(* CODESYS project 2019-30-07-Sparkplug_Commands.ecp

Project tree, tasks and I/O mapping:
  PFC_Sparkplug : 750-8212 PFC200 2ETH RS, WAGO, order no. 0750-8212, version 5.13.2.32
    application Application
      libraries: ; WagoAppCloud, 1.3.0.8 (WAGO)
      task PLC_Task (cyclic, interval t#100ms, priority 15) calls PLC_PRG
      program PLC_PRG [ST]
      program VariableLogger [ST]
      program CommandHandler [ST]
      function block FbChangeOfValue_Real [ST]
      function block FbChangeOfValue_Byte [ST]
      function block FbChangeOfValue_Bool [ST]
    Kbus : Kbus, WAGO, version 1.4.0.2
        unmapped channels: K-BUS diagnostics
    MODBUS
      MODBUS : MODBUS, WAGO, order no. n/a, version 1.1.1.15
    Serial
      COM1 : COM1, WAGO, version 0.0.0.19
    Common.PCI
*)

// PFC_Sparkplug/Application/PLC_PRG
(* Purpose of the example program: Communicate with a Sparkplug primary application *)
PROGRAM PLC_PRG

CommandHandler();
VariableLogger();

END_PROGRAM

// PFC_Sparkplug/Application/CommandHandler
(* Purpose of the example program: Receive and handle commands aka "metric-change-requests" from the Sparkplug primary application
Ignition has functionality for "write tag", so within the commands our example program will define exacly one parameter,
which is actually the writable metric from ignitions point of view. 
The data protocol Sparkplug doesn't support response messages. (FbCommandResponse) *)
PROGRAM CommandHandler
VAR
	(* Use the function block FbCommandConfigurator to send the command configuration to the cloud *)
	oFbCmdConfigurator : 	WagoAppCloud.FbCommandConfigurator;
	(* Define two commands in the list *)
	aCommandDescriptions : 	ARRAY [0..1] OF WagoAppCloud.typCommandDescription;

	(*	Listen to command calls from the cloud using the FbCommandListener.
	It will set the xCommandReceived flag to true if a command is called. *)
	oFbCmdHandler : WagoAppCloud.FbCommandListener;
	xCommandReceived: BOOL;
	IncomingCommand : WagoAppCloud.typCommandRequest;
	dwReceivedCmdId : DWORD;

	(* Parameter to get the received value from the cloud *)
	rParameter1 : REAL;
	sParameter2 : STRING;
END_VAR

(* Init command1 and its Request Parameter *)		
aCommandDescriptions[0].bCommandId := 1;
aCommandDescriptions[0].bNumberOfRequestParameters := 1;
aCommandDescriptions[0].bNumberOfResponseParameters := 0;	(* The data protocol Sparkplug doesn't support response messages. This is an information for Wago Protocol. *)
aCommandDescriptions[0].sName := 'MyFirstCommand';
aCommandDescriptions[0].aRequestParameters[0].sParameterName := 'Parameter 1 from Cloud to PFC';
aCommandDescriptions[0].aRequestParameters[0].eParameterType := WagoAppCloud.eCommandParameterType.CPT_REAL;

(* Init command2 and its Request Parameter *)		
aCommandDescriptions[1].bCommandId := 2;
aCommandDescriptions[1].bNumberOfRequestParameters := 1;
aCommandDescriptions[1].bNumberOfResponseParameters := 0;
aCommandDescriptions[1].sName := 'MySecondCommand';
aCommandDescriptions[1].aRequestParameters[0].sParameterName := 'Parameter 2 from Cloud to PFC';
aCommandDescriptions[1].aRequestParameters[0].eParameterType := WagoAppCloud.eCommandParameterType.CPT_STRING;

(* Configurate the commands and send the commands configuration to the cloud *)
oFbCmdConfigurator(	pSupportedCommands := ADR(aCommandDescriptions),
					bNumberOfSupportedCommands := 2);

(* Receive data to get the command from the cloud *)
oFbCmdHandler(pCommand:= ADR(IncomingCommand), 
				xCommandReceived=> xCommandReceived);

(* Handle command *)
IF xCommandReceived THEN
	dwReceivedCmdId := IncomingCommand.dwCommandId;

	CASE dwReceivedCmdId OF
		1:
			(* received command with the command ID 1 *)
			rParameter1 := STRING_TO_REAL(IncomingCommand.aRequestParameters[0].sParameterValue);
			
		2:
			(* received command with the command ID 2 *)
			sParameter2 := IncomingCommand.aRequestParameters[0].sParameterValue;
	END_CASE
END_IF

END_PROGRAM

// PFC_Sparkplug/Application/VariableLogger
PROGRAM VariableLogger

VAR
	(* Some value to transfer *)
	iVariable1 		: INT 	:= -32768;
	dwVariable2		: DWORD := 7;
	lrVariable3		: LREAL	:= 21.53;

	bVariable4		: BYTE 	:= 255;
	xVariable5		: BOOL := FALSE;
	rVariable6		: REAL 	:= 1.234;	
	
	wVariable7		: WORD	:= 49;
	iVariable8		: INT 	:= -32768;
	
	(* Define 3 collections *)
	aCollections	: ARRAY[0..2] OF WagoAppCloud.typCollection;

	(* Define 3 variable descriptions for the collections *)
	aVariableDescriptions1	: ARRAY[0..2] OF WagoAppCloud.typVariableDescription;
	aVariableDescriptions2	: ARRAY[0..2] OF WagoAppCloud.typVariableDescription;
	aVariableDescriptions3	: ARRAY[0..1] OF WagoAppCloud.typVariableDescription;
	
	tSampleInterval1		: TIME := T#10S;
	tMinPublishInterval		: TIME := T#0S; (* choose the smallest possible publish interval *)
	
	oFbCollectionLogger		: WagoAppCloud.FbCollectionLogger;
END_VAR

VAR
	oFbChangeOfValue		: FbChangeOfValue_Bool;
	oFbChangeOfValue_Real	: FbChangeOfValue_Real;
	oFbChangeOfValue_Byte	: FbChangeOfValue_Byte;
	
	(* Timer *)
	xEnableTimer: BOOL := TRUE;
	tCyclicTimerSendTagCollection: TON;
END_VAR

(* Simulate changing values to transfer to the cloud *)
	iVariable1 := iVariable1 + 3;
	dwVariable2 := dwVariable2 + 100;
	lrVariable3 := lrVariable3 - 1234.12;
	bVariable4 := bVariable4 + 2;
	IF bVariable4 > 150 THEN
		xVariable5 := TRUE;
	ELSE
		xVariable5 := FALSE;
	END_IF
	rVariable6 := rVariable6 + 100;
	wVariable7 := wVariable7 + 1;
	iVariable8 := iVariable8 + 1;

(* Configuration of the collections and variables *)
	
(* Init and configure collection 1 *)
	aVariableDescriptions1[0].pAddress := ADR(iVariable1);
	aVariableDescriptions1[0].eValueType := WagoAppCloud.VVT_INT;
	aVariableDescriptions1[0].sTag := 'var1_int';
	aVariableDescriptions1[0].sUnit := 'u1';
	
	aVariableDescriptions1[1].pAddress := ADR(dwVariable2);
	aVariableDescriptions1[1].eValueType := WagoAppCloud.VVT_DWORD;
	aVariableDescriptions1[1].sTag := 'var2_dword';
	aVariableDescriptions1[1].sUnit := 'u2';
	
	aVariableDescriptions1[2].pAddress := ADR(lrVariable3);
	aVariableDescriptions1[2].eValueType := WagoAppCloud.VVT_LREAL;
	aVariableDescriptions1[2].sTag := 'var3_lreal';
	aVariableDescriptions1[2].sUnit := 'u3';
	
	aCollections[0].dwCollectionId := 1;
	aCollections[0].sName := 'MyFirstCollection';
	aCollections[0].pVariableDescriptions := ADR(aVariableDescriptions1);
	aCollections[0].dwVariablesCount := 3;
	(* Configuration of the mode to sampling the data. 
	In this case the samples of collection 1 will be set automatically. The space between two timestamps are defined in the sample interval. *)
	aCollections[0].eSamplingDataMode := eSamplingMode.LIBRARY_DEFAULT_AUTOMATIC;		(* LIBRARY_DEFAULT_AUTOMATIC is the default mode *)
	aCollections[0].pSampleInterval := ADR(tSampleInterval1);
	aCollections[0].pPublishInterval := ADR(tMinPublishInterval);

(* Init and configure collection 2 *)
	aVariableDescriptions2[0].pAddress := ADR(bVariable4);
	aVariableDescriptions2[0].eValueType := WagoAppCloud.VVT_BYTE;
	aVariableDescriptions2[0].sTag := 'var4_byte';
	aVariableDescriptions2[0].sUnit := 'u3';
	
	aVariableDescriptions2[1].pAddress := ADR(xVariable5);
	aVariableDescriptions2[1].eValueType := WagoAppCloud.VVT_BOOL;
	aVariableDescriptions2[1].sTag := 'var5_bool';
	aVariableDescriptions2[1].sUnit := 'u4';
	
	aVariableDescriptions2[2].pAddress := ADR(rVariable6);
	aVariableDescriptions2[2].eValueType := WagoAppCloud.VVT_REAL;
	aVariableDescriptions2[2].sTag := 'var6_real';
	aVariableDescriptions2[2].sUnit := 'u5';
	
	aCollections[1].dwCollectionId := 2;
	aCollections[1].sName := 'MySecondCollection';
	aCollections[1].pVariableDescriptions := ADR(aVariableDescriptions2);
	aCollections[1].dwVariablesCount := 3;
	(* Configuration of the mode to sampling the data. 
	In this case the samples of collection 2 will be set manual by the PLC application. 
	The Trigger of a sample is set manual with the CollectionTrigger or the VariableTrigger.
	
	Note for data protocol Sparkplug: The sampling mode UNEQUALLY_SPACED_CUSTOMIZED_SAMPLES will be used for all manual generatted samples. 
	Sampling modes UNEQUALLY_SPACED_COLLECTION_SAMPLES, EQUALLY_SPACED_COLLECTION_SAMPLES, EQUALLY_SPACED_CUSTOMIZED_SAMPLES are not needed for Sparkplug. 
	This differentation between the different manual generatted sample modes is only an interesting information for the Wago Protocol. *)
	aCollections[1].eSamplingDataMode := eSamplingMode.UNEQUALLY_SPACED_CUSTOMIZED_SAMPLES; 
	aCollections[1].pPublishInterval := ADR(tMinPublishInterval);
	
(* Init and cnfigure collection 3 *)
	aVariableDescriptions3[0].pAddress := ADR(wVariable7);
	aVariableDescriptions3[0].eValueType := WagoAppCloud.VVT_WORD;
	aVariableDescriptions3[0].sTag := 'var7_word';
	aVariableDescriptions3[0].sUnit := 'u3';
	
	aVariableDescriptions3[1].pAddress := ADR(iVariable8);
	aVariableDescriptions3[1].eValueType := WagoAppCloud.VVT_INT;
	aVariableDescriptions3[1].sTag := 'var8_int';
	aVariableDescriptions3[1].sUnit := 'u4';
	
	aCollections[2].dwCollectionId := 3;
	aCollections[2].sName := 'MyThirdCollection';
	aCollections[2].pVariableDescriptions := ADR(aVariableDescriptions3);
	aCollections[2].dwVariablesCount := 2;
	(* Configuration of the mode to sampling the data. 
	In this case the samples of collection 3 will be set manual by the PLC application. 
	The Trigger of a sample is set manual with the CollectionTrigger or the VariableTrigger. 
	
	Note for data protocol Sparkplug: The sampling mode UNEQUALLY_SPACED_CUSTOMIZED_SAMPLES will be used for all manual generatted samples. 
	Sampling modes UNEQUALLY_SPACED_COLLECTION_SAMPLES, EQUALLY_SPACED_COLLECTION_SAMPLES, EQUALLY_SPACED_CUSTOMIZED_SAMPLES are not needed for Sparkplug. 
	This differentation between the different manual generatted sample modes is only an interesting information for the Wago Protocol. *)
	aCollections[2].eSamplingDataMode := eSamplingMode.UNEQUALLY_SPACED_CUSTOMIZED_SAMPLES;
	aCollections[2].pPublishInterval := ADR(tMinPublishInterval);

(* Example to set the event if variable value exceeded the threshold values - Variable Trigger*)
oFbChangeOfValue_Byte(	bInput:= bVariable4,
						bActivate:= 100,
						bDeactivate:= 70,
						xTrigger:= aVariableDescriptions2[0].xVariableTrigger);

oFbChangeOfValue(	xVariable:= xVariable5, 
					xTrigger:= aVariableDescriptions2[1].xVariableTrigger);

oFbChangeOfValue_Real(	rInput:= rVariable6, 
						rActivate:= 1500,
						rDeactivate:= 700,
						xTrigger:= aVariableDescriptions2[2].xVariableTrigger);

(* Example to set the event with a timer intervall - CollectionTrigger or VariableTrigger *)
(* Set an event with an Timer to send the variables in an intervall to the cloud *)
tCyclicTimerSendTagCollection(IN:= xEnableTimer, PT:= T#30S);

IF tCyclicTimerSendTagCollection.Q THEN
	aCollections[1].xCollectionTrigger := TRUE;
	aCollections[2].xCollectionTrigger := TRUE;

	xEnableTimer := FALSE;
ELSE
	xEnableTimer := TRUE;
END_IF
						
oFbCollectionLogger(pCollections := ADR(aCollections),
					dwCollectionsCount := 3);

END_PROGRAM

// PFC_Sparkplug/Application/FbChangeOfValue_Bool
FUNCTION_BLOCK FbChangeOfValue_Bool
VAR_INPUT
	xVariable : BOOL; 	(* Input value *)
END_VAR
VAR_IN_OUT
	xTrigger : BOOL; 	(* Variable Trigger - trigger is set only once when the value was changed and reset with the function block WagoAppCloud.FbCollectionLogger *)
END_VAR
VAR
	xLastSendedState : BOOL := FALSE; 	(* save the old value when this value was sending to the cloud to the if the value was changing *)
END_VAR

IF NOT xTrigger THEN
	IF NOT (xVariable = xLastSendedState) THEN
		xTrigger := TRUE;
		xLastSendedState := xVariable;
	END_IF
END_IF

END_FUNCTION_BLOCK

// PFC_Sparkplug/Application/FbChangeOfValue_Real
(* The function block FbChangeOfValue_Real shows an example how an event of a real variable could be triggered.
*)

FUNCTION_BLOCK FbChangeOfValue_Real

VAR_INPUT
	rInput 		: REAL;
	rActivate 	: REAL;
	rDeactivate : REAL;
END_VAR

VAR_IN_OUT
	xTrigger	: BOOL;
END_VAR

VAR
	xLastSendedState : BOOL := FALSE;
END_VAR

IF NOT xTrigger THEN
	IF rActivate > rDeactivate THEN
		IF (rInput >= rActivate) AND NOT xLastSendedState THEN
			xTrigger := TRUE;
			xLastSendedState := TRUE;
		ELSIF (rInput <= rDeactivate) AND xLastSendedState THEN
			xTrigger := TRUE;
			xLastSendedState := FALSE;
		END_IF
	ELSE
		IF (rInput <= rActivate) AND NOT xLastSendedState THEN
			xTrigger := TRUE;
			xLastSendedState := TRUE;
		ELSIF (rInput >= rDeactivate) AND xLastSendedState THEN
			xTrigger := TRUE;
			xLastSendedState := FALSE;
		END_IF
	END_IF
END_IF

END_FUNCTION_BLOCK

// PFC_Sparkplug/Application/FbChangeOfValue_Byte
(* The function block FbChangeOfValue_Byte shows an example how an event of a real variable could be triggered.
*)

FUNCTION_BLOCK FbChangeOfValue_Byte

VAR_INPUT
	bInput 		: BYTE; (* Input value *)
	bActivate 	: BYTE; (* Threshold value at which the output signal is set to TRUE *)
	bDeactivate : BYTE; (* Threshold value at which the output signal is set to FALSE *)
END_VAR

VAR_IN_OUT
	xTrigger	: BOOL; (* VariableTrigger - trigger is set only once when the value was changed and reset with the function block WagoAppCloud.FbCollectionLogger *)
END_VAR

VAR
	xLastSendedState : BOOL := FALSE; (* state of the last sended changed state - send a change only once when the threshold was exceeded *)
END_VAR

(* Do only something when the VariableTrigger isn't activated (the VariableTrigger will be reset by the function block FbCollectionLogger) *)
IF NOT xTrigger THEN
	(* Two variations are to be considered during the analysis of the input values *)
	
	(* case 1: the activate threshold is greater as the deactivate threshold *)	
	IF bActivate > bDeactivate THEN
		(* rising edge *)
		IF (bInput >= bActivate) AND NOT xLastSendedState THEN
			xTrigger := TRUE;
			xLastSendedState := TRUE;
		(* falling edge *)
		ELSIF (bInput <= bDeactivate) AND xLastSendedState THEN
			xTrigger := TRUE;
			xLastSendedState := FALSE;
		END_IF
		
	(* case 2: the deactivate threshold is greater as the activate threshold *)
	ELSE
		(* rising edge *)
		IF (bInput <= bActivate) AND NOT xLastSendedState THEN
			xTrigger := TRUE;
			xLastSendedState := TRUE; (* save that the trigger after the rising edge is already set so that the trigger will be only set once *)
		(* falling edge *)
		ELSIF (bInput >= bDeactivate) AND xLastSendedState THEN
			xTrigger := TRUE;
			xLastSendedState := FALSE;
		END_IF
	END_IF
END_IF

END_FUNCTION_BLOCK
